TYPE DigitalOutput :
STRUCT
	out AT %Q*	:	BIT;
END_STRUCT
END_TYPE

(* stored: Version 1.1.0.1, ProductVersion 3.1.4020.12
   DUT DigitalOutput: Id {8a5a2876-bec8-4fdd-8f1c-2a3713d30f9e} *)
